// TIA Portal project "Proyecto - Esqueleto" (V19)

(* hardware
DEVICE "S7-1200 station_1"  S7-1200 Station
   slot 0: "Rack_0"  S7-1200 Rack  Rack  V1.0
   slot 1: "PLC_1"  CPU 1214C DC/DC/DC  6ES7 214-1AG40-0XB0  V4.6
DEVICE "HMI_2"  KTP400 Basic mono PN
   slot 0: "HMI_2"  KTP400 Basic mono PN  6AV6 647-0AA11-3AX0  12.0.0.0
   slot 1: "HMI_RT_2"  KTP400 Basic mono PN  6AV6 647-0AA11-3AX0  12.0.0.0
   slot 5: "HMI_2.IE_CP_1"  PROFINET Interface  12.0.0.0
      slot 1: "PROFINET Interface_1"  PROFINET Interface
         slot 1: "Port_1"  Port
*)

// ===== PLC "PLC_1"  CPU 1214C DC/DC/DC =====

ORGANIZATION_BLOCK "Main"   // OB1, LAD, ProgramCycle
TITLE = "Main Program Sweep (Cycle)"
{ S7_Optimized_Access := 'TRUE' }
VERSION : 0.1
   VAR_INPUT
      Initial_Call : Bool;   // Initial call of this OB
      Remanence : Bool;   // =True, if remanent data are available
   END_VAR
BEGIN
END_ORGANIZATION_BLOCK

(* ===== HMI "HMI_RT_2" =====
system functions are stored by id; their names below are inferred from use
connection "HMI_Connection_1": ETHERNET, SMART_S7_1200_OMS

HMI tags "Default tag table"
   "Tag_ScreenNumber" : UInt, internal

Template "Template_1" 320x240
   Button "Exit" at 249,202 size 52x37; TextOff 'Exit'; PictureOff "ExitRuntime_KTP400_Basic_mono_PN"; PictureOn "ExitRuntime_KTP400_Basic_mono_PN"
      on Release: StopRuntime(0)
   Button "Template_Button" at 175,202 size 52x37; TextOff 'Text'
   Button "Alarms" at 101,202 size 52x37; TextOff 'Alarms'; PictureOff "AlarmDisplay_KTP400_Basic_mono_PN"; PictureOn "AlarmDisplay_KTP400_Basic_mono_PN"
      on Release: function_ef3f5d25("Alarm window_Unacknowledged", -1)
   Button "Start screen" at 27,202 size 52x37; TextOff 'Start screen'; PictureOff "NavigateHome_KTP400_Basic_mono_PN"; PictureOn "NavigateHome_KTP400_Basic_mono_PN"
      on Release: ActivateScreen("Root screen", 0)
   SymbolicIOField "Symbolic_IO_Field_Screen" at 69,7 size 164x24; TextOff '0'; TextOn '1'; TextList "TextList_ScreenNames"
      ProcessValue <- "Tag_ScreenNumber"
      on Change: ActivateScreenByNumber("Tag_ScreenNumber", 0)
   DateTimeField "HmiScreenItemData" at 235,19 size 85x19
   DateTimeField "HmiScreenItemData_1" at 235,0 size 85x19
   GraphicView "Logo" at 0,0 size 67x38; Picture "Logo of HMI_2"

screen "Root screen" 320x240, template "Template_1"
   on GenerateScreen: SetTag("Tag_ScreenNumber", 1)
   TextField "HmiScreenItemData" at 32,99 size 256x36; Text 'Welcome to HMI_2 (KTP400 Basic mono PN)!'
*)